(*!
<summary>Provides the mutable reset capability of an exception.</summary>
<description>
Extends IReadOnlyException with Clear. Clearing changes this exception state; it neither transfers ownership
nor grants permission to delete task-managed snapshots. Consumers that only inspect errors should use
IReadOnlyException.
</description>
*)
(*
SPDX-FileCopyrightText: © 2026 Oleksandr Tiutyk <trofimich@gmail.com>
SPDX-License-Identifier: MIT
License: https://opensource.org/license/mit
*)

INTERFACE IException EXTENDS IReadOnlyException

(*!
<summary>Clears diagnostic state for reuse without deleting this instance.</summary>
<description>
Does not extend the lifetime of borrowed references or transfer ownership. Concrete implementations define
which metadata is reset; disposal calls must not raise exceptions.
</description>
*)

METHOD Clear
END_METHOD

END_INTERFACE

(* stored: Version 1.1.0.1
   Itf IException: Id {0a7624ed-9c88-4373-b895-6c0f3e6612e5}
   Method Clear: Id {3fb14633-892d-4442-b75e-6b5e593146ae} *)
